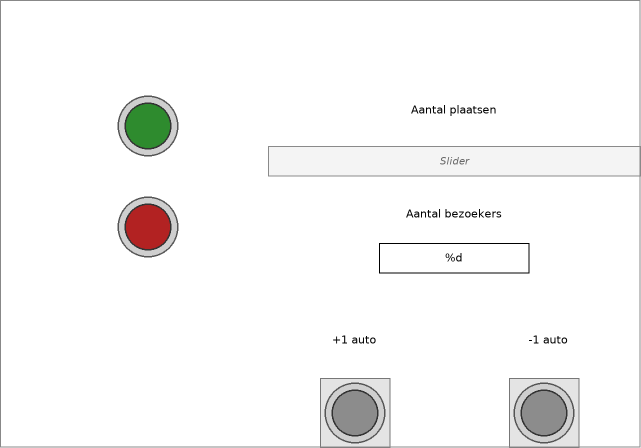
VISUALIZATION Visualization  // 641x448
    Slider (268,146 373x30), variable: MAIN.iAantalplaatsen, scale 0..100
    Rectangle (379,243 150x30), "%d", text variable: MAIN.iTellerstand, invisible if: MAIN.iTellerstand
        p4168582468: MAIN.iTellerstand
    Label (379,199 150x30), "Aantal bezoekers"
    Label (379,95 150x30), "Aantal plaatsen"
    Lamp1 (113,192 70x70), variable: MAIN.bRood, style: Lamp-Lamp1-Red
    Lamp1 (113,91 70x70), variable: MAIN.bGroen, style: Lamp-Lamp1-Green
    PushSwitch (320,378 70x70), variable: MAIN.Plus1auto, behaviour: TOGGLE, style: Switch-PushSwitch-Gray
    PushSwitch (509,378 70x70), variable: MAIN.Min1auto, behaviour: TOGGLE, style: Switch-PushSwitch-Gray
    Label (279,325 150x30), "+1 auto"
    Label (473,325 150x30), "-1 auto"
END_VISUALIZATION

(* stored: Version 1.1.0.1, ProductVersion 3.1.4024.12
   Visu Visualization: Id {e1a6c678-8e80-4f06-8255-5e79a8d744a3} *)
